Fanuc KAREL source: KO00143.KL

PROGRAM KO00143
%NOLOCKGROUP
VAR
  R: REAL
  CFG: CONFIG
  OUT: XYZWPR
  N: ARRAY[2] OF BYTE
BEGIN
  N[1] = 1
  R = 2.0
  CFG.CFG_FLIP = TRUE
  OUT = POS(R, R, R, N[1], R, R, CFG)
END KO00143
